// TIA Portal V21 export
// export: Created 2026-07-28T22:13:03.2791291Z, ExportSetting WithDefaults, DisplayName Totally Integrated Automation Portal, DisplayVersion V21, DisplayName SINAMICS Startdrive Advanced, DisplayVersion V21, DisplayName SINAMICS Startdrive G110M, G120, G120C, G120D, G120P, G115D, DisplayVersion V21, DisplayName SINAMICS Startdrive G130, G150, S120, S150, G200, G220, S200, S210, S220, Innomotics MVD, DisplayVersion V21, DisplayName STEP 7 Professional, DisplayVersion V21, DisplayName STEP 7 Safety, DisplayVersion V21, DisplayName Tech WebApplication, DisplayVersion V21, DisplayName WinCC Basic/Comfort/Advanced, DisplayVersion V21, DisplayName WinCC Professional, DisplayVersion V21, DisplayName WinCC Unified, DisplayVersion V21
VAR_GLOBAL   // PLC tag table "MOTOR_AREA_01 (MOTOR_01)"
   MOTOR_01_RESERVA_01 AT %M5512.0 : Bool;
   MOTOR_01_RESERVA_02 AT %M5512.1 : Bool;
   MOTOR_01_RESERVA_DINT_01 AT %MD5513 : DInt;
   "MOTOR_01_STS_HABILITA_IMPAR_&" AT %M5506.4 : Bool;   // Status: Condições para partida do equipamento MOTOR_01 estão OK
   MOTOR_01_FALHA AT %M5500.7 : Bool;   // Status: Falha geral do equipamento MOTOR_01
   MOTOR_01_STS_FALHA_NAO_LIGOU AT %M5506.1 : Bool;   // Status: Falha de partida do equipamento MOTOR_01
   MOTOR_01_CMD_HABILITA_LIGA_AUTO2 AT %M5500.2 : Bool;   // Comando: Habilitação para partida em modo automático para o equipamento MOTOR_01
   MOTOR_01_SP_SETPOINT_AUTO AT %MW5502 : Int;   // Setpoint: Valor de referência em modo automático para o equipamento MOTOR_01
   "MOTOR_01_STS_HABILITA_PAR_&" AT %M5506.5 : Bool;   // Status: Condições para partida do equipamento MOTOR_01 estão OK
   MOTOR_01_CMD_BOTAO_RESET_FALHA AT %M5500.0 : Bool;   // Comando: Botão de reset de falhas para o equipamento MOTOR_01
   MOTOR_01_STS_VAR_MONITORADA AT %MD5508 : Real;   // Status: Variável monitorada (Ex: vibração, temperatura) do equipamento MOTOR_01
   MOTOR_01_STS_REMOTO_AUTO AT %M5507.3 : Bool;   // Status: Comando Remoto em modo Automático para o equipamento MOTOR_01
   MOTOR_01_STS_REMOTO_MANUAL AT %M5507.4 : Bool;   // Status: Comando Remoto em modo Manual para o equipamento MOTOR_01
   MOTOR_01_STS_LIGADO_PROFINET AT %M5506.6 : Bool;   // Status: Comunicação Profinet OK com o equipamento MOTOR_01
   MOTOR_01_STS_ALTERNANCIA_OK AT %M5506.0 : Bool;   // Tag de controle/status/falha para o equipamento MOTOR_01
   MOTOR_01_CMD_RESET_LIGA AT %M5500.6 : Bool;   // Comando: Reset do comando Ligar o equipamento MOTOR_01
   MOTOR_01_CMD_RESET_FALHA_PROFINET AT %M5500.5 : Bool;   // Comando: Reset de falha Profinet para o equipamento MOTOR_01
   MOTOR_01_STS_MODO_REMOTO AT %M5507.2 : Bool;   // Status: Chave seletora do equipamento MOTOR_01 em Remoto
   MOTOR_01_LIGADO AT %M5501.0 : Bool;   // Status: Equipamento MOTOR_01 em operação
   MOTOR_01_CMD_HABILITA_LIGA_AUTO AT %M5500.1 : Bool;   // Comando: Habilitação para partida em modo automático para o equipamento MOTOR_01
   MOTOR_01_STS_LOCAL_MANUAL AT %M5507.0 : Bool;   // Status: Comando Local em modo Manual para o equipamento MOTOR_01
   MOTOR_01_STS_FALHA_PROFINET AT %M5506.2 : Bool;   // Status: Falha de comunicação Profinet com o equipamento MOTOR_01
   MOTOR_01_STS_SUCCAO_OK AT %M5507.5 : Bool;   // Status: Condição de sucção OK para a bomba MOTOR_01
   MOTOR_01_STS_MODO_LOCAL AT %M5507.1 : Bool;   // Status: Chave seletora do equipamento MOTOR_01 em Local
   MOTOR_01_STS_HABILITA AT %M5506.3 : Bool;   // Status: Condições para partida do equipamento MOTOR_01 estão OK
   MOTOR_01_STS_LOCAL_AUTO AT %M5506.7 : Bool;   // Status: Comando Local em modo Automático para o equipamento MOTOR_01
   MOTOR_01_CMD_LIGA_PROFINET AT %M5500.4 : Bool;   // Comando: Partida via Profinet para o equipamento MOTOR_01
   MOTOR_01_SP_SETPOINT_MANUAL AT %MW5504 : Int;   // Setpoint: Valor de referência em modo manual para o equipamento MOTOR_01
   MOTOR_01_CMD_LIGA_BOMBA AT %M5500.3 : Bool;   // Comando: Ligar/Partir a bomba MOTOR_01
END_VAR
